FUNCTION_BLOCK Load4Station
VAR_INPUT
END_VAR
VAR_OUTPUT
END_VAR
VAR
	xTrigger :BOOL := FALSE; // triggers processing
	State : eLoadSta4State := eLoadSta4State.eUnknown;
	NextState : eLoadSta4State := eLoadSta4State.eUnknown;
	bFirst : BOOL := TRUE;
	VUT : BYTE; //VehicleID Under Station
	DwellTimer : TON;
	LoadingComplete : BOOL := FALSE;
	CycleNumb: INT := 0;
	RowNumber :INT:=0;
	SeedNumber : INT:=1;
END_VAR

IF (GVL_IO.MachineEStopped) THEN 
	State := eLoadSta4State.eUnknown;
	NextState := eLoadSta4State.eUnknown;
END_IF

CASE State OF

eLoadSta4State.eUnknown:
	NextState := eLoadSta4State.eReady;

eLoadSta4State.eInit:

eLoadSta4State.eHoming:

eLoadSta4State.eReady:

	IF (xTrigger) THEN
		NextState := eLoadSta4State.eWaitForLoadComplete;
		
		DwellTimer(IN:=FALSE);		
	END_IF

eLoadSta4State.eDwell:


eLoadSta4State.eWaitForLoadComplete:
	 IF (LoadingComplete) THEN
		NextState := eLoadSta4State.eDepart;
		UpdatePartData();
		LoadingComplete := FALSE;
		DwellTimer(IN:=FALSE);
	END_IF
	
eLoadSta4State.eProcessing:


eLoadSta4State.eDepart:
	Stations.fbRoutePlanner.M_NotifyVehStaCmpl(StationIndex:= MM_CONST.LOAD_4_STA, VehicleID := VUT);
	xTrigger := FALSE;
    IF (Stations.fbCycleControl.StopRequested) THEN
		NextState := eLoadSta4State.eStopActive;
	ELSE	
		NextState := eLoadSta4State.eReady;	
	END_IF

eLoadSta4State.eStopActive:
	IF (NOT Stations.fbCycleControl.StopRequested) THEN
		NextState := eLoadSta4State.eReady;
	END_IF

eLoadSta4State.eError:

END_CASE

IF (State <> NextState) THEN
	bFirst := TRUE;
ELSE
	bFirst := FALSE;
END_IF

State := NextState;
Status.StationsState[MM_CONST.LOAD_4_STA_HMI_STATE] := State;

METHOD PUBLIC ClearVehicleTrigger : BOOL
VAR_INPUT
END_VAR
xTrigger := FALSE;
END_METHOD

PROPERTY PUBLIC LoadComplete : BOOL
SET
LoadingComplete := LoadComplete;
END_SET
END_PROPERTY

METHOD PUBLIC ResetState : BOOL
VAR_INPUT
END_VAR
	State := eLoadSta4State.eUnknown;
	NextState := eLoadSta4State.eUnknown;
END_METHOD

METHOD PUBLIC SetRowNumber : BOOL
VAR_INPUT
	RowLocationNumber : INT;
END_VAR
RowNumber := RowLocationNumber;
END_METHOD

PROPERTY PUBLIC Trigger : BOOL
SET
xTrigger := Trigger;
END_SET
END_PROPERTY

METHOD PUBLIC UpdatePartData : BOOL
VAR_INPUT
END_VAR
memset(ADR(PartsData.Status[VUT]),0,SIZEOF(PartDataType));
PartsData.Status[VUT].LoadTime := SYSTEMTIME_TO_STRING(Logging.fbCurrTime.systemTime);
//PartsData.Status[VUT].CavityNumber := 13 + (CycleNumb MOD 4);
PartsData.Status[VUT].CavityNumber := RowNumber + SeedNumber;
CycleNumb := CycleNumb+1; // Use this till Yushin Robot sends out this information with Bit Location ID
PartsData.Status[VUT].OverallStatus := ePartStatus.eLoaded; // At least that is the assumption. We may want to check on how to turn off cavities later, but this will be caught by vision.
PartsData.Status[VUT].BarrelSize := LotsData.Lot.BarrelSize; // we are copying this data in case we might in future want to have more than one lots running at the same time on the machine
PartsData.Status[VUT].PartNumber := LotsData.Lot.PartNumber; // we are copying this data in case we might in future want to have more than one lots running at the same time on the machine
PartsData.Status[VUT].LotNumber := LotsData.Lot.LotNumber; // we are copying this data in case we might in future want to have more than one lots running at the same time on the machine
END_METHOD

PROPERTY PUBLIC VehicleUnderTest : BYTE
GET
VehicleUnderTest := VUT;
END_GET
SET
VUT := VehicleUnderTest;
END_SET
END_PROPERTY

END_FUNCTION_BLOCK

(* stored: Version 1.1.0.1, ProductVersion 3.1.4022.3
   POU Load4Station: Id {7a5f58c4-4a71-40f0-bb29-10f5624d8fc7}, SpecialFunc None
   Method ClearVehicleTrigger: Id {98324f79-9da3-46f6-bb5a-ee98087427e2}
   Property LoadComplete: Id {38483af5-d682-4f0a-b45d-5a6e7dd8801f}
   Set Set: Id {585a7733-b4b7-419b-819f-d7b14b63950f}
   Method ResetState: Id {092af0ca-d838-4202-bdc5-3b60db42d280}
   Method SetRowNumber: Id {727445d8-daa3-448a-95e9-5252fb26b5b7}
   Property Trigger: Id {5ea3908a-a725-4710-88a3-33e2ff35bebf}
   Set Set: Id {d9c9462e-68f2-4479-a604-d9e870ecfeea}
   Method UpdatePartData: Id {a44c1ff4-47d6-4eda-845b-1530edd6d866}
   Property VehicleUnderTest: Id {6a0e2e28-7606-43ed-8aa4-9124c532ff0c}
   Get Get: Id {78054811-cff8-4830-b046-9fdb999766c9}
   Set Set: Id {09b44ece-f5e9-43ef-9aaf-1fa3c99a4957} *)
